(* PLC project PLC1, Unknown Unnamed 1 *)
(* stored: creationDateTime 2021-02-24T14:42:08, modificationDateTime 2024-06-25T11:48:42 *)

FUNCTION_BLOCK SUB_0
  VAR_INPUT
    IN1 : DINT;
  END_VAR
  VAR_OUTPUT
    real_value : DINT;
  END_VAR
  VAR
    i : DINT;
    exc : __SYSTEM.ExceptionCode;
  END_VAR

            __TRY
real_value := IN1 - 5;
IN1 := 5/IN1;
__CATCH(exc)
i:=IN1;
  while i<5 do
    real_value:= 6;
    i:=i*i;
  end_while;
__ENDTRY;
          
END_FUNCTION_BLOCK

PROGRAM PLC3
  VAR_INPUT
    level : DINT;
  END_VAR
  VAR_OUTPUT
    pump : BOOL;
  END_VAR
  VAR
    low : BOOL;
    real_value : DINT;
    high : BOOL;
    low_3 : DINT := 0;
    high_3 : DINT := 10;
    SUB_00 : SUB_0;
  END_VAR

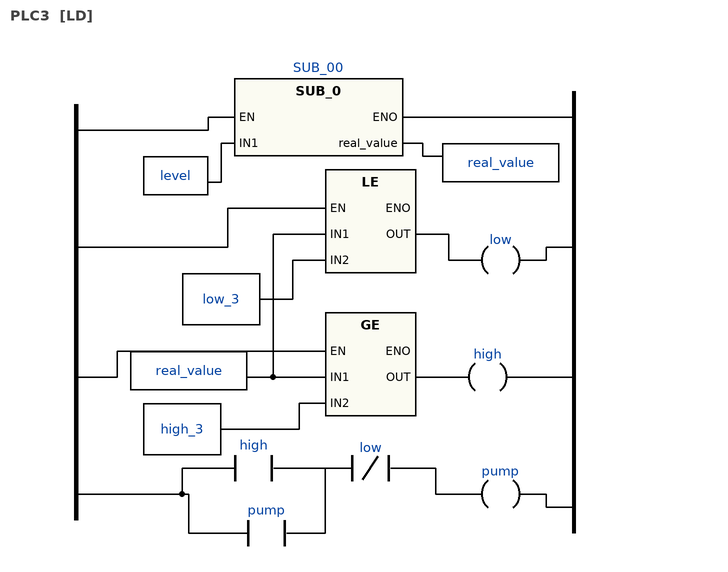
(* LD diagram, written out as Structured Text *)
high := real_value >= high_3;
low := real_value <= low_3;
pump := (high OR pump) AND NOT low;
SUB_00(IN1 := level);
real_value := SUB_00.real_value;
END_PROGRAM

PROGRAM PLC2
  VAR_INPUT
    level : DINT;
  END_VAR
  VAR_OUTPUT
    request : BOOL;
  END_VAR
  VAR
    open_req : BOOL;
    close_req : BOOL;
    low_2 : DINT := 10;
    high_2 : DINT := 20;
  END_VAR

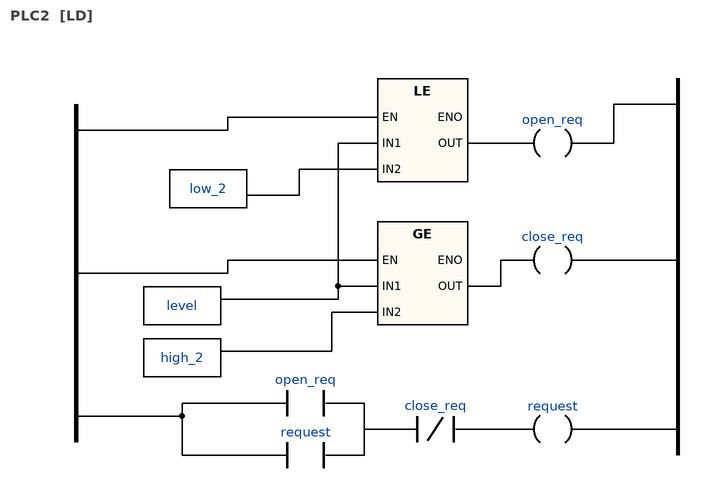
(* LD diagram, written out as Structured Text *)
close_req := level >= high_2;
open_req := level <= low_2;
request := (open_req OR request) AND NOT close_req;
END_PROGRAM

PROGRAM PLC1
  VAR_INPUT
    level : DINT;
    request : DINT;
  END_VAR
  VAR_OUTPUT
    pumps : BOOL;
    valve : BOOL;
  END_VAR
  VAR
    low : BOOL;
    high : BOOL;
    open_req : BOOL;
    close_req : BOOL;
    low_1 : DINT := 40;
    high_1 : DINT := 80;
  END_VAR

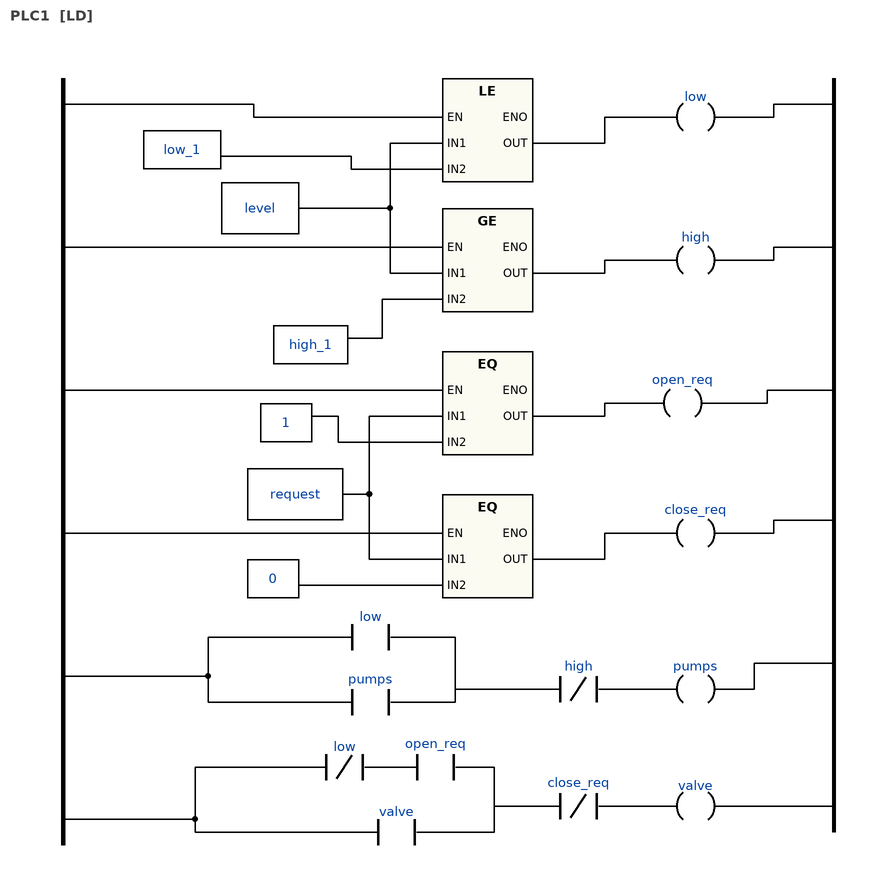
(* LD diagram, written out as Structured Text *)
low := level <= low_1;
high := level >= high_1;
pumps := (low OR pumps) AND NOT high;
valve := (NOT low AND open_req OR valve) AND NOT close_req;
open_req := request = 1;
close_req := request = 0;
END_PROGRAM

CONFIGURATION Config0
  RESOURCE Res0 ON PLC
    TASK task0(INTERVAL := T#20ms, PRIORITY := 0);
    TASK task1(INTERVAL := T#20ms, PRIORITY := 0);
    TASK task2(INTERVAL := T#20ms, PRIORITY := 0);
    PROGRAM instance0 WITH task0 : PLC1;
    PROGRAM instance1 WITH task1 : PLC2;
    PROGRAM instance2 WITH task2 : PLC3;
  END_RESOURCE
END_CONFIGURATION
